FUNCTION INTERNAL Power2 : LREAL
VAR_INPUT
  v : LREAL;
END_VAR

Power2 := v*v;

END_FUNCTION

(* stored: Version 1.1.0.1
   POU Power2: Id {0e3e86d0-3b11-44f2-b301-06ab88dcd5f9}, SpecialFunc None *)
